// TIA Portal project "Project1" (V17)

(* hardware
DEVICE "S7-1200 station_1"  S7-1200 Station
   slot 0: "Rack_0"  S7-1200 Rack  Rack  V1.0
   slot 1: "PLC_1"  CPU 1214C AC/DC/Rly  6ES7 214-1BG31-0XB0  V3.0
DEVICE "HMI_1"  KTP600 Basic color PN
   slot 0: "HMI_1"  KTP600 Basic color PN  6AV6 647-0AD11-3AX0  12.0.0.0
   slot 1: "HMI_RT_1"  KTP600 Basic color PN  6AV6 647-0AD11-3AX0  12.0.0.0
   slot 5: "HMI_1.IE_CP_1"  PROFINET Interface  12.0.0.0
      slot 1: "PROFINET Interface_1"  PROFINET Interface
         slot 1: "Port_1"  Port
DEVICE "S7-1200 station_2"  S7-1200 Station
   slot 0: "Rack_0"  S7-1200 Rack  Rack  V1.0
   slot 1: "PLC_2"  CPU 1214C DC/DC/DC  6ES7 214-1AG40-0XB0  V4.5
*)

// ===== PLC "PLC_1"  CPU 1214C AC/DC/Rly =====

VAR_GLOBAL   // PLC tag table "Default tag table"
   "Pieza al inicio de la cinta" AT %I0.0 : Bool;
   "Pieza en el centro de la cinta" AT %I0.1 : Bool;
   "Pieza al final de la cinta" AT %I0.2 : Bool;
   "Carro retraido" AT %I0.4 : Bool;
   "Carro avanzado" AT %I0.5 : Bool;
   "Ventosa en parte superior" AT %I0.6 : Bool;
   "Pieza succionada" AT %I0.7 : Bool;
   "Avance de la cinta" AT %Q0.0 : Bool;
   "Retroceso de la cinta" AT %Q0.1 : Bool;
   "Avance del separador" AT %Q0.2 : Bool;
   "Retroceso del carro" AT %Q0.4 : Bool;
   "Avance del carro" AT %Q0.5 : Bool;
   "Ventosa en la parte inferior" AT %Q0.6 : Bool;
   "Conexión de vacio" AT %Q0.7 : Bool;
   "Inicio" AT %M0.0 : Bool;
   "Pausa" AT %M0.1 : Bool;
   "MPS Inicio" AT %M0.2 : Bool;
END_VAR

// folder: System blocks/Program resources

DATA_BLOCK "IEC_Timer_0_DB_3"   // DB4
{ S7_Optimized_Access := 'TRUE' }
AUTHOR : Simatic
FAMILY : IEC
NAME : IEC_TMR
VERSION : 1.0
// stored: InstanceOfName IEC_TIMER
"IEC_TIMER"
BEGIN
END_DATA_BLOCK

// folder: (top level)

ORGANIZATION_BLOCK "Main"   // OB1, LAD, ProgramCycle
TITLE = "Main Program Sweep (Cycle)"
{ S7_Optimized_Access := 'TRUE' }
VERSION : 0.1
   VAR_TEMP
      Temp_1 : Bool;
   END_VAR
BEGIN

REGION Network 1
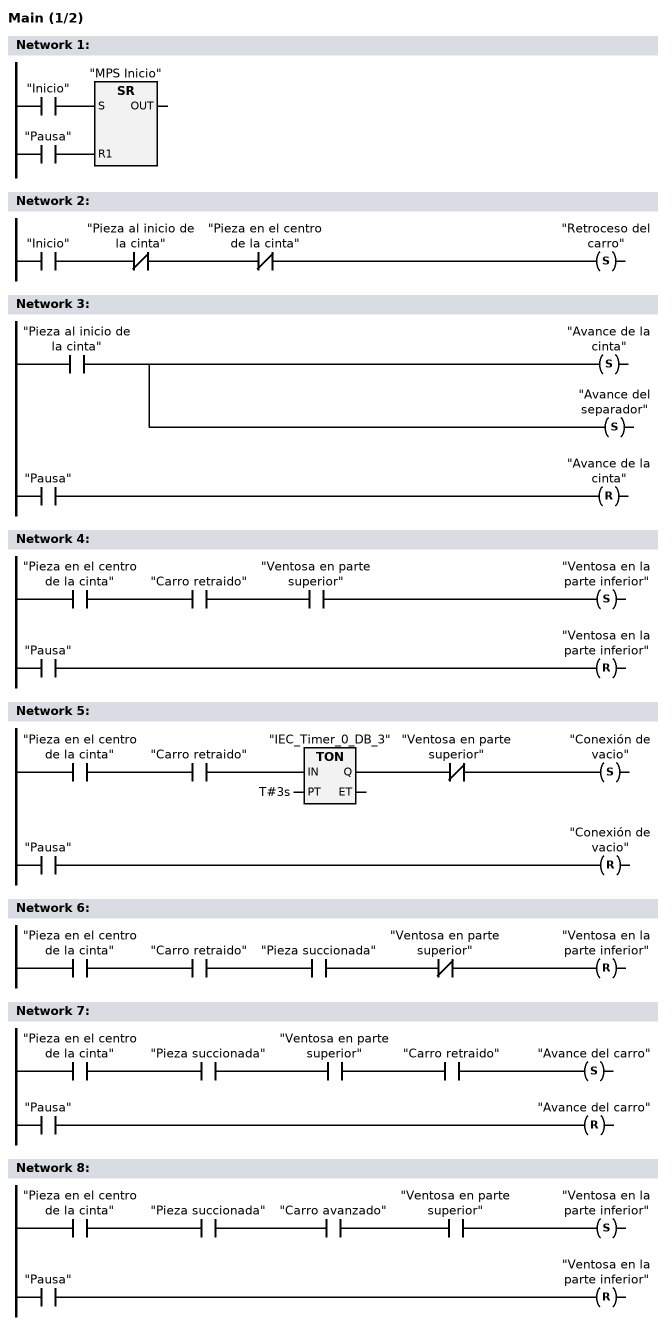
   RUNG wire#powerrail
      Contact( "Inicio" )
      S_SR(operand := "MPS Inicio", r1 := wire#w1)
   END_RUNG
   RUNG wire#powerrail
      Contact( "Pausa" )
   END_RUNG wire#w1
   // the same network as SCL:
   IF "Inicio" THEN
       "MPS Inicio" := TRUE;   // SR flip-flop
   END_IF;
   IF "Pausa" THEN "MPS Inicio" := FALSE; END_IF;
END_REGION

REGION Network 2
   RUNG wire#powerrail
      Contact( "Inicio" )
      I_Contact( "Pieza al inicio de la cinta" )
      I_Contact( "Pieza en el centro de la cinta" )
      S_Coil( "Retroceso del carro" )
   END_RUNG
   // the same network as SCL:
   IF "Inicio" AND NOT "Pieza al inicio de la cinta" AND NOT "Pieza en el centro de la cinta" THEN
       "Retroceso del carro" := TRUE;
   END_IF;
END_REGION

REGION Network 3
   RUNG wire#powerrail
      Contact( "Pieza al inicio de la cinta" )
      wire#w1
      S_Coil( "Avance de la cinta" )
   END_RUNG
   RUNG wire#w1
      S_Coil( "Avance del separador" )
   END_RUNG
   RUNG wire#powerrail
      Contact( "Pausa" )
      R_Coil( "Avance de la cinta" )
   END_RUNG
   // the same network as SCL:
   IF "Pieza al inicio de la cinta" THEN
       "Avance de la cinta" := TRUE;
       "Avance del separador" := TRUE;
   END_IF;
   IF "Pausa" THEN "Avance de la cinta" := FALSE; END_IF;
END_REGION

REGION Network 4
   RUNG wire#powerrail
      Contact( "Pieza en el centro de la cinta" )
      Contact( "Carro retraido" )
      Contact( "Ventosa en parte superior" )
      S_Coil( "Ventosa en la parte inferior" )
   END_RUNG
   RUNG wire#powerrail
      Contact( "Pausa" )
      R_Coil( "Ventosa en la parte inferior" )
   END_RUNG
   // the same network as SCL:
   IF "Pieza en el centro de la cinta" AND "Carro retraido" AND "Ventosa en parte superior" THEN
       "Ventosa en la parte inferior" := TRUE;
   END_IF;
   IF "Pausa" THEN "Ventosa en la parte inferior" := FALSE; END_IF;
END_REGION

REGION Network 5
   "IEC_Timer_0_DB_3".TON(IN := "Pieza en el centro de la cinta" AND "Carro retraido", PT := T#3s);
   IF "IEC_Timer_0_DB_3".Q AND NOT "Ventosa en parte superior" THEN "Conexión de vacio" := TRUE; END_IF;
   IF "Pausa" THEN "Conexión de vacio" := FALSE; END_IF;
END_REGION

REGION Network 6
   RUNG wire#powerrail
      Contact( "Pieza en el centro de la cinta" )
      Contact( "Carro retraido" )
      Contact( "Pieza succionada" )
      I_Contact( "Ventosa en parte superior" )
      R_Coil( "Ventosa en la parte inferior" )
   END_RUNG
   // the same network as SCL:
   IF "Pieza en el centro de la cinta" AND "Carro retraido" AND "Pieza succionada" AND NOT "Ventosa en parte superior" THEN
       "Ventosa en la parte inferior" := FALSE;
   END_IF;
END_REGION

REGION Network 7
   RUNG wire#powerrail
      Contact( "Pieza en el centro de la cinta" )
      Contact( "Pieza succionada" )
      Contact( "Ventosa en parte superior" )
      Contact( "Carro retraido" )
      S_Coil( "Avance del carro" )
   END_RUNG
   RUNG wire#powerrail
      Contact( "Pausa" )
      R_Coil( "Avance del carro" )
   END_RUNG
   // the same network as SCL:
   IF "Pieza en el centro de la cinta" AND "Pieza succionada" AND "Ventosa en parte superior" AND "Carro retraido" THEN
       "Avance del carro" := TRUE;
   END_IF;
   IF "Pausa" THEN "Avance del carro" := FALSE; END_IF;
END_REGION

REGION Network 8
   RUNG wire#powerrail
      Contact( "Pieza en el centro de la cinta" )
      Contact( "Pieza succionada" )
      Contact( "Carro avanzado" )
      Contact( "Ventosa en parte superior" )
      S_Coil( "Ventosa en la parte inferior" )
   END_RUNG
   RUNG wire#powerrail
      Contact( "Pausa" )
      R_Coil( "Ventosa en la parte inferior" )
   END_RUNG
   // the same network as SCL:
   IF "Pieza en el centro de la cinta" AND "Pieza succionada" AND "Carro avanzado" AND "Ventosa en parte superior" THEN
       "Ventosa en la parte inferior" := TRUE;
   END_IF;
   IF "Pausa" THEN "Ventosa en la parte inferior" := FALSE; END_IF;
END_REGION

REGION Network 9
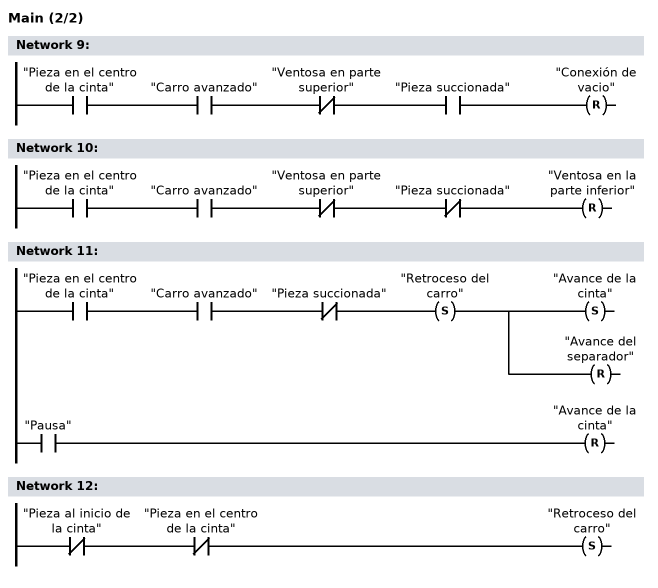
   RUNG wire#powerrail
      Contact( "Pieza en el centro de la cinta" )
      Contact( "Carro avanzado" )
      I_Contact( "Ventosa en parte superior" )
      Contact( "Pieza succionada" )
      R_Coil( "Conexión de vacio" )
   END_RUNG
   // the same network as SCL:
   IF "Pieza en el centro de la cinta" AND "Carro avanzado" AND NOT "Ventosa en parte superior" AND "Pieza succionada" THEN
       "Conexión de vacio" := FALSE;
   END_IF;
END_REGION

REGION Network 10
   RUNG wire#powerrail
      Contact( "Pieza en el centro de la cinta" )
      Contact( "Carro avanzado" )
      I_Contact( "Ventosa en parte superior" )
      I_Contact( "Pieza succionada" )
      R_Coil( "Ventosa en la parte inferior" )
   END_RUNG
   // the same network as SCL:
   IF "Pieza en el centro de la cinta" AND "Carro avanzado" AND NOT "Ventosa en parte superior" AND NOT "Pieza succionada" THEN
       "Ventosa en la parte inferior" := FALSE;
   END_IF;
END_REGION

REGION Network 11
   RUNG wire#powerrail
      Contact( "Pieza en el centro de la cinta" )
      Contact( "Carro avanzado" )
      I_Contact( "Pieza succionada" )
      S_Coil( "Retroceso del carro" )
      wire#w1
      S_Coil( "Avance de la cinta" )
   END_RUNG
   RUNG wire#w1
      R_Coil( "Avance del separador" )
   END_RUNG
   RUNG wire#powerrail
      Contact( "Pausa" )
      R_Coil( "Avance de la cinta" )
   END_RUNG
   // the same network as SCL:
   IF "Pieza en el centro de la cinta" AND "Carro avanzado" AND NOT "Pieza succionada" THEN
       "Retroceso del carro" := TRUE;
       "Avance de la cinta" := TRUE;
       "Avance del separador" := FALSE;
   END_IF;
   IF "Pausa" THEN "Avance de la cinta" := FALSE; END_IF;
END_REGION

REGION Network 12
   RUNG wire#powerrail
      I_Contact( "Pieza al inicio de la cinta" )
      I_Contact( "Pieza en el centro de la cinta" )
      S_Coil( "Retroceso del carro" )
   END_RUNG
   // the same network as SCL:
   IF NOT "Pieza al inicio de la cinta" AND NOT "Pieza en el centro de la cinta" THEN
       "Retroceso del carro" := TRUE;
   END_IF;
END_REGION
END_ORGANIZATION_BLOCK

// ===== PLC "PLC_2"  CPU 1214C DC/DC/DC =====

VAR_GLOBAL   // PLC tag table "Default tag table"
   "Pieza al inicio de la cinta" AT %I0.0 : Bool;
   "Pieza en el centro de la cinta" AT %I0.1 : Bool;
   "Pieza al final de la cinta" AT %I0.2 : Bool;
   "Carro retraido" AT %I0.4 : Bool;
   "Carro avanzado" AT %I0.5 : Bool;
   "Ventosa en parte superior" AT %I0.6 : Bool;
   "Pieza succionada" AT %I0.7 : Bool;
   "Avance de la cinta" AT %Q0.0 : Bool;
   "Retroceso de la cinta" AT %Q0.1 : Bool;
   "Avance del separador" AT %Q0.2 : Bool;
   "Retroceso del separador" AT %Q0.3 : Bool;
   "Retroceso del carro" AT %Q0.4 : Bool;
   "Avance del carro" AT %Q0.5 : Bool;
   "Ventosa en la parte inferior" AT %Q0.6 : Bool;
   "Conexión de vacio" AT %Q0.7 : Bool;
   "Inicio Mps" AT %M0.2 : Bool;
   "Inicio" AT %M0.0 : Bool;
   "Pausa" AT %M0.1 : Bool;
END_VAR

// folder: System blocks/Program resources

DATA_BLOCK "IEC_Timer_0_DB"   // DB1
{ S7_Optimized_Access := 'TRUE' }
AUTHOR : Simatic
FAMILY : IEC
NAME : IEC_TMR
VERSION : 1.0
// stored: InstanceOfName IEC_TIMER
"IEC_TIMER"
BEGIN
END_DATA_BLOCK

DATA_BLOCK "IEC_Timer_0_DB_1"   // DB2
{ S7_Optimized_Access := 'TRUE' }
AUTHOR : Simatic
FAMILY : IEC
NAME : IEC_TMR
VERSION : 1.0
// stored: InstanceOfName IEC_TIMER
"IEC_TIMER"
BEGIN
END_DATA_BLOCK

DATA_BLOCK "IEC_Timer_0_DB_2"   // DB3
{ S7_Optimized_Access := 'TRUE' }
AUTHOR : Simatic
FAMILY : IEC
NAME : IEC_TMR
VERSION : 1.0
// stored: InstanceOfName IEC_TIMER
"IEC_TIMER"
BEGIN
END_DATA_BLOCK

DATA_BLOCK "IEC_Timer_0_DB_3"   // DB4
{ S7_Optimized_Access := 'TRUE' }
AUTHOR : Simatic
FAMILY : IEC
NAME : IEC_TMR
VERSION : 1.0
// stored: InstanceOfName IEC_TIMER
"IEC_TIMER"
BEGIN
END_DATA_BLOCK

// folder: (top level)

ORGANIZATION_BLOCK "Main"   // OB1, LAD, ProgramCycle
TITLE = "Main Program Sweep (Cycle)"
{ S7_Optimized_Access := 'TRUE' }
VERSION : 0.1
   VAR_INPUT
      Initial_Call : Bool;   // Initial call of this OB
      Remanence : Bool;   // =True, if remanent data are available
   END_VAR
   VAR_TEMP   // added for the SCL form of the ladder/FBD networks
      _w1 : Bool;
   END_VAR
BEGIN

REGION Network 1
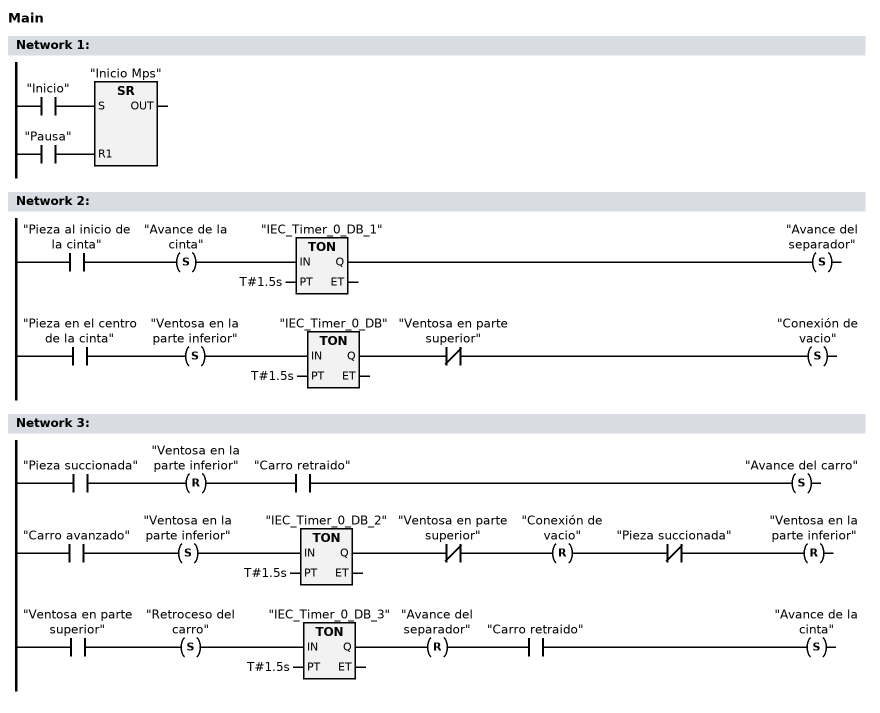
   RUNG wire#powerrail
      Contact( "Inicio" )
      S_SR(operand := "Inicio Mps", r1 := wire#w1)
   END_RUNG
   RUNG wire#powerrail
      Contact( "Pausa" )
   END_RUNG wire#w1
   // the same network as SCL:
   IF "Inicio" THEN
       "Inicio Mps" := TRUE;   // SR flip-flop
   END_IF;
   IF "Pausa" THEN "Inicio Mps" := FALSE; END_IF;
END_REGION

REGION Network 2
   IF "Pieza al inicio de la cinta" THEN "Avance de la cinta" := TRUE; END_IF;
   "IEC_Timer_0_DB_1".TON(IN := "Pieza al inicio de la cinta", PT := T#1.5s);
   IF "IEC_Timer_0_DB_1".Q THEN "Avance del separador" := TRUE; END_IF;
   IF "Pieza en el centro de la cinta" THEN "Ventosa en la parte inferior" := TRUE; END_IF;
   "IEC_Timer_0_DB".TON(IN := "Pieza en el centro de la cinta", PT := T#1.5s);
   IF "IEC_Timer_0_DB".Q AND NOT "Ventosa en parte superior" THEN "Conexión de vacio" := TRUE; END_IF;
END_REGION

REGION Network 3
   IF "Pieza succionada" THEN "Ventosa en la parte inferior" := FALSE; END_IF;
   IF "Pieza succionada" AND "Carro retraido" THEN "Avance del carro" := TRUE; END_IF;
   IF "Carro avanzado" THEN "Ventosa en la parte inferior" := TRUE; END_IF;
   "IEC_Timer_0_DB_2".TON(IN := "Carro avanzado", PT := T#1.5s);
   #_w1 := "IEC_Timer_0_DB_2".Q AND NOT "Ventosa en parte superior";
   IF #_w1 THEN "Conexión de vacio" := FALSE; END_IF;
   IF #_w1 AND NOT "Pieza succionada" THEN "Ventosa en la parte inferior" := FALSE; END_IF;
   IF "Ventosa en parte superior" THEN "Retroceso del carro" := TRUE; END_IF;
   "IEC_Timer_0_DB_3".TON(IN := "Ventosa en parte superior", PT := T#1.5s);
   IF "IEC_Timer_0_DB_3".Q THEN "Avance del separador" := FALSE; END_IF;
   IF "IEC_Timer_0_DB_3".Q AND "Carro retraido" THEN "Avance de la cinta" := TRUE; END_IF;
END_REGION
END_ORGANIZATION_BLOCK

(* ===== HMI "HMI_RT_1" =====
system functions are stored by id; their names below are inferred from use
connection "HMI_Connection_1": ETHERNET, SMART_S7_1200_OMS

HMI tags "Default tag table"
   "Inicio" : Bool = PLC Inicio AT %M0.0, 1 s
   "Pausa" : Bool = PLC Pausa AT %M0.1, 1 s

Template "Template_1" 320x240
   Button "Exit" at 266,202 size 52x37; TextOff 'Exit'; PictureOff "ExitRuntime_KTP600_Basic_color_PN"; PictureOn "ExitRuntime_KTP600_Basic_color_PN"
      on Release: StopRuntime(0)
   Button "Template_Button" at 213,202 size 52x37; TextOff 'Text'
   Button "Template_Button_1" at 160,202 size 52x37; TextOff 'Text'
   Button "Template_Button_2" at 107,202 size 52x37; TextOff 'Text'
   Button "Alarms" at 54,202 size 52x37; TextOff 'Alarms'; PictureOff "AlarmDisplay_KTP600_Basic_color_PN"; PictureOn "AlarmDisplay_KTP600_Basic_color_PN"
      on Release: function_ef3f5d25("Alarm window_Unacknowledged", -1)
   Button "Start screen" at 1,202 size 52x37; TextOff 'Start screen'; PictureOff "NavigateHome_KTP600_Basic_color_PN"; PictureOn "NavigateHome_KTP600_Basic_color_PN"
      on Release: ActivateScreen("Root screen", 0)
   DateTimeField "HmiScreenItemData" at 235,19 size 85x19
   DateTimeField "HmiScreenItemData_1" at 235,0 size 85x19
   GraphicView "Logo" at 0,0 size 67x38; Picture "Logo of HMI_1"

screen "Root screen" 320x240, template "Template_1"
   on GenerateScreen: SetTag("Inicio", 1)
   Button "Button_1" at 28,96 size 96x32; TextOff 'Inicio'
      on Press: SetBit("Inicio")
      on Release: SetBit("Inicio")
   Button "Button_2" at 186,96 size 96x32; TextOff 'Pausa'
      on Press: SetBit("Pausa")
      on Release: SetBit("Pausa")
   TextField "Text field_1" at 88,10 size 124x16; Text 'Pick & Place Station'
*)